{attribute 'qualified_only'}
{attribute 'strict'}
TYPE EXAMPLE_ENUM :
(
	Example0 := 0,
	Example1 := 1,
	Example2 := 2
);
END_TYPE

(* stored: Version 1.1.0.1, ProductVersion 3.1.4022.10
   EnumerationTextList EXAMPLE_ENUM: Id {9299cb57-e6ee-4651-b1a2-ac58ac99f0ae} *)
